TYPE ST_InputsSickScanner_CLV690 :
STRUCT	
	CtrlIn					: ST_CtrlInSickScanner;
	ConfMessageIn			: ARRAY[0..31] OF BYTE; // Message Byte 5 and forward result from scanner			
	Heartbeat				: BOOL;	
	GoodRead				: BOOL; 				//Good read signal from scanner	
END_STRUCT
END_TYPE

(* stored: Version 1.1.0.1, ProductVersion 3.1.4024.4
   DUT ST_InputsSickScanner_CLV690: Id {793bacfd-1cee-4764-b079-0f64be2eef34} *)
